{region '#Template'}
	{attribute 'Version' := '5.0.0.0'}
	{attribute 'Tags' := '"LCID": "1031", "Text": "Fassade, Sonnenschutz, Thermoautomatik"'}
	{attribute 'Tags' := '"LCID": "1033", "Text": "Facade, Sunprotection, thermoautomatic"'}
	{attribute 'Using' := '"Type": "Template", "URI": "ST_BA_SunBld"'}
	{attribute 'Using' := '"Type": "Template", "URI": "E_BA_SunBldPrio"'}
	{attribute 'Description' := '"LCID": "1031", "Text": "Sonnenschutz fassadenweite Thermoautomatik"'}
	{attribute 'Description' := '"LCID": "1033", "Text": "Sunprotection facade-thermoautomatic"'}
{endregion}
FUNCTION_BLOCK FB_BA_Facade_ThermoAutomatic EXTENDS FB_BA_View
VAR_INPUT
	bFcdInSun				: BOOL;	
	fRefRmT					: REAL;
	fRefRmTCol				: REAL;
	fRefRmTHtg				: REAL;	
END_VAR                 	
VAR_OUTPUT              	
	stSunBld				: ST_BA_SunBld;
	bThAutoEvent			: BOOL;
	                    	
END_VAR                 	
VAR_INPUT CONSTANT      	
	FcdThAutoEn				: FB_BA_BV_Op;		
	FcdThAutoColPos			: FB_BA_AV_Op;		
	FcdThAutoColAngl		: FB_BA_AV_Op;		
	FcdThAutoEvent			: FB_BA_SunBldEvt			:=(ePrio:=E_BA_SunBldPrio.eFacadeThermoAutomatic);			
END_VAR                 	
VAR                     	
	FcdThAutoHtgCol			: FB_BA_Swi2P;
	bFcdThAuto_Enable		: BOOL;
	fFcdThAuto_Position		: REAL;
	fFcdThAuto_Angle		: REAL;
END_VAR
VAR // added by the converter: edge detectors and wires of the graphical bodies
    _w1 : BOOL;
END_VAR

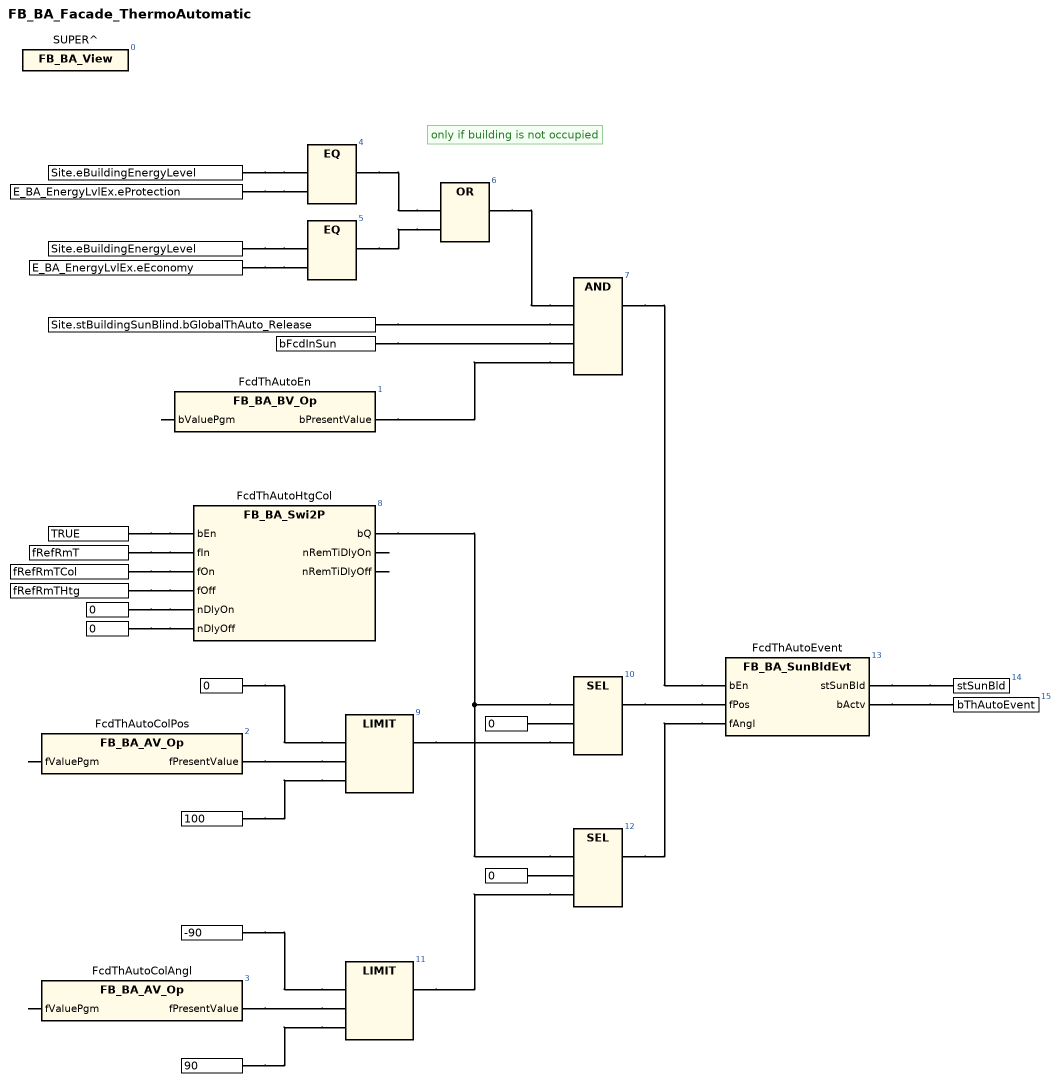
SUPER^(); // FB_BA_View
FcdThAutoEn(); // FB_BA_BV_Op
FcdThAutoColPos(); // FB_BA_AV_Op
FcdThAutoColAngl(); // FB_BA_AV_Op
// only if building is not occupied
_w1 := (Site.eBuildingEnergyLevel = E_BA_EnergyLvlEx.eProtection OR Site.eBuildingEnergyLevel = E_BA_EnergyLvlEx.eEconomy) AND Site.stBuildingSunBlind.bGlobalThAuto_Release AND bFcdInSun AND FcdThAutoEn.bPresentValue;
FcdThAutoHtgCol(
    bEn := TRUE,
    fIn := fRefRmT,
    fOn := fRefRmTCol,
    fOff := fRefRmTHtg,
    nDlyOn := 0,
    nDlyOff := 0); // FB_BA_Swi2P
FcdThAutoEvent(
    bEn := _w1,
    fPos := SEL(FcdThAutoHtgCol.bQ, 0, LIMIT(0, FcdThAutoColPos.fPresentValue, 100)),
    fAngl := SEL(FcdThAutoHtgCol.bQ, 0, LIMIT(-90, FcdThAutoColAngl.fPresentValue, 90))); // FB_BA_SunBldEvt
stSunBld := FcdThAutoEvent.stSunBld;
bThAutoEvent := FcdThAutoEvent.bActv;

METHOD FB_init : BOOL
VAR_INPUT
	bInitRetains : BOOL; // if TRUE; the retain variables are initialized (warm start / cold start)
	bInCopyCode : BOOL;  // if TRUE; the instance afterwards gets moved into the copy code (online change)
END_VAR
FcdThAutoEn.iParent				:= THIS^;
FcdThAutoEn.iLabel				:= LblCtl_FacadeThermoAutomaticEnable;
FcdThAutoEn.sObjectName		   	:= '{Idx=01}';
FcdThAutoEn.sInactiveText		:= txtEvent_Off;
FcdThAutoEn.sActiveText			:= txtEvent_On;
FcdThAutoEn.bValueRm			:= FALSE;
FcdThAutoEn.eToggleMode			:= E_BA_ToggleMode.eSwitch;        
                            	
                            	
FcdThAutoColPos.iParent			:= THIS^;  
FcdThAutoColPos.iLabel			:= LblCtl_FacadeThermoAutomaticCoolingPosition;	
FcdThAutoColPos.sObjectName		:= '{Idx=01}';
FcdThAutoColPos.eUnit			:= E_BA_Unit.eOther_Percent; 
FcdThAutoColPos.fValueRm		:= 100.0;
                            	
		                    	
FcdThAutoColAngl.iParent		:= THIS^;
FcdThAutoColAngl.iLabel			:= LblCtl_FacadeThermoAutomaticCoolingAngle;	
FcdThAutoColAngl.sObjectName	:= '{Idx=02}';
FcdThAutoColAngl.eUnit			:= E_BA_Unit.eOther_DegreesAngular; 
FcdThAutoColAngl.fValueRm		:= -90.0;
END_METHOD

END_FUNCTION_BLOCK

(* stored: Version 1.1.0.1, ProductVersion 3.1.4024.12
   POU FB_BA_Facade_ThermoAutomatic: Id {b5820f81-b109-488b-95d7-57aec38a7581}, SpecialFunc None
   Method FB_init: Id {abd50743-6a99-4687-b5b8-7cdc3b88a9db} *)
